# EPICS substitutions: mc01/tpmacApp/pmc/xf23id2-mc01-homing.substitutions
file "home_to_enc_ref_template.pmc"
{

pattern
{ AXIS,   PLC,  SERVO,  TIMER }
{ 1,      8,    701,    5511  }
{ 2,      9,    702,    5512  }
{ 3,      10,    703,    5611  }
{ 4,      11,    704,    5612  }

}

file "home_to_limit_template.pmc"
{

pattern
{ AXIS,   PLC,  SERVO,  TIMER }
{ 8,      15,    714,    5812  }

}
